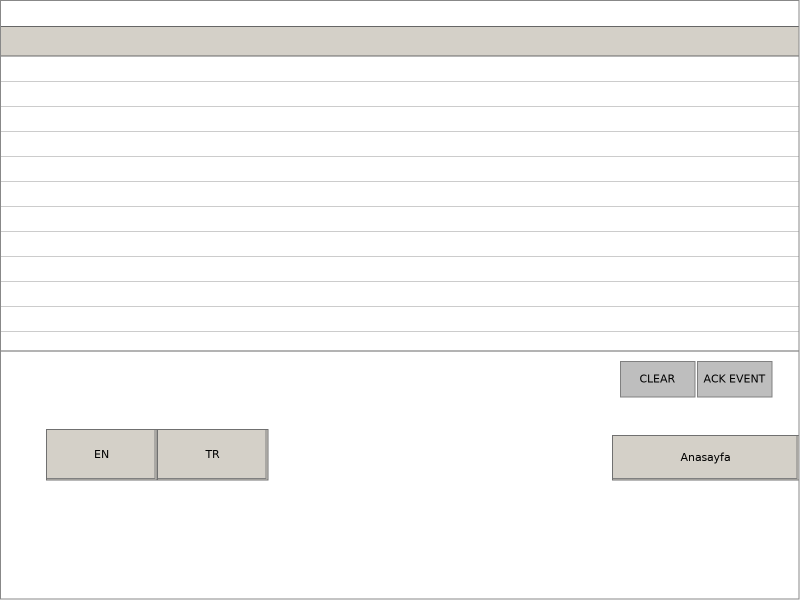
VISUALIZATION VISU_1910_PlcEvents  // 800x600
    Table (0,26 799x325), data array: stEvents.Plc.stEventsVisu
        p3854506369: stEvents.Plc.stEventsVisu[INDEX].nEventType
        p1892666644: stEvents.Plc.stEventsVisu[INDEX].nEventID
        p338671338: stEvents.Plc.stEventsVisu[INDEX].nEventColor
        p2170511999: stEvents.Plc.stEventsVisu[INDEX].nTextColor
        p3723444502: stEvents.Plc.stEventsVisu[INDEX].sEventTime
        p1218418051: stEvents.Plc.stEventsVisu[INDEX].sEventAckTime
        p2232123230: Event Type
        p2237128397: Event Time
        p505689113: Ack Time
        p1420305297: stEvents.Plc.nTableSelX
        p1137915858: stEvents.Plc.nTableSelY
        p1128707560: nPlcEventsNumber
        Columns.Column.[0].Template: stEvents.Plc.nFrameColor
        Columns.Column.[1].Template: stEvents.Plc.nFrameColor
        Columns.Column.[4].Template: stEvents.Plc.nFrameColor
        Columns.Column.[5].Template: stEvents.Plc.nFrameColor
    Rectangle (697,361 75x36), "ACK EVENT", colour toggle: stEvents.Plc.bAckEvent
        tap stEvents.Plc.bAckEvent
    Rectangle (620,361 75x36), "CLEAR", colour toggle: stEvents.Plc.bClearEventTable
        tap stEvents.Plc.bClearEventTable
    Button (612,435 187x45), "Anasayfa"
        OnMouseClick: change screen: Visualization
    Button (46,429 111x51), "EN"
        OnMouseClick: ChangeLanguage ChangeLanguage=English
    Button (157,429 111x51), "TR"
        OnMouseClick: ChangeLanguage ChangeLanguage=Turkish
END_VISUALIZATION

(* stored: Version 1.1.0.1, ProductVersion 3.1.4024.12
   Visu VISU_1910_PlcEvents: Id {5d6740cd-06ab-4e29-8b23-da43c1a21c20} *)
